Universal Robots PolyScope program: RC_E8_PLACE_831.urp

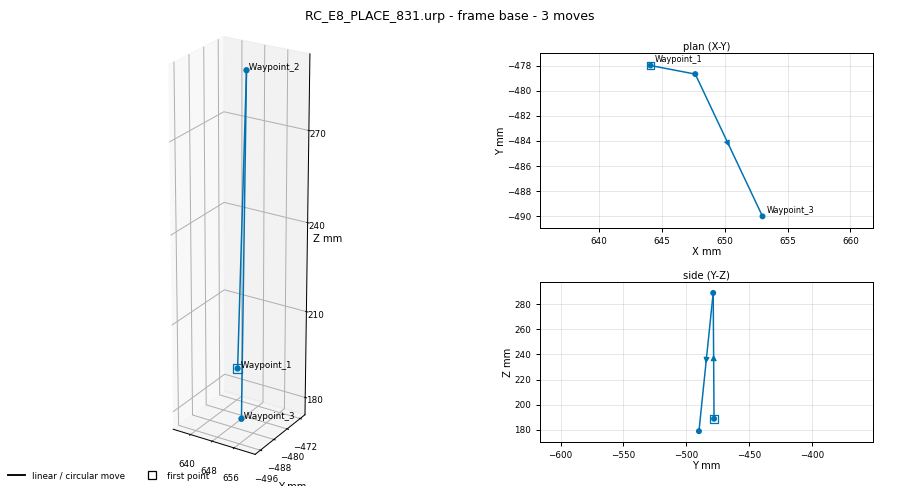
[picture p0: tool path of RC_E8_PLACE_831.urp in frame base, 3 of 3 moves have a stored position in this frame; points joined in program order, loops and branches not executed]
Program RC_E8_PLACE_831 (createdIn=3.0.0 lastSavedIn=3.0.0 directory=/programs installation=default)
Robot Program (runOnlyOnce=true motionType=MoveJ speed=1.047198 acceleration=1.396263 useActiveTCP=false)
  'Program generated by RoboDK v4.1.0 for UR3e_HORNO on 06/09/2022 17:07:52'
  'Using nominal kinematics.'
  'Using Ref. Frame Traslado C: p[0.369000, -0.220000, 0.032000, 0.000000, 0.000000, 0.000000]'
  'Using TCP 0208-0001-0001-307-000-3 Horno: p[0.000000, 0.000000, 0.164750, 0.000000, 0.000000, 0.000000]'
  Script: set_tcp(p[0.000000, 0.000000, 0.164750, 0.000000, 0.000000, 0.000000])
  Script: movej([-0.418006, -2.151118, -0.151320, -2.416408, 1.600991, 4.345870],0.60000,0.12500,0,0.0000)
  MoveL speed 100 mm/s, acceleration 120 mm/s^2 (useActiveTCP=true)
    Waypoint Waypoint_1: TCP in base x=644.083 y=-478 z=188.872 mm, rx=3.1385 ry=-0.0805 rz=-0.0117 rad; joints [-22.639, -103.728, -69.335, -97.291, 89.736, 250.301] deg; flange x=645.315 y=-477.69 z=353.617 mm, rx=3.1385 ry=-0.0805 rz=-0.0117 rad
  'Detach from 0208-0001-0001-307-000-3 Horno'
  MoveL speed 500 mm/s, acceleration 900 mm/s^2 (useActiveTCP=true)
    Waypoint Waypoint_2: TCP in base x=647.647 y=-478.682 z=288.936 mm, rx=-3.1102 ry=0.0802 rz=-0.0087 rad; joints [-23.95, -123.25, -8.67, -138.45, 91.73, 249] deg; flange x=646.6 y=-483.659 z=453.608 mm, rx=-3.1102 ry=0.0802 rz=-0.0087 rad
  Script: movej([-0.418006, -2.151118, -0.151320, -2.416408, 1.600991, 4.345870],0.90000,0.50000,0,0.0000)
  Script: movej([0.453224, -1.802935, -0.994995, -3.455038, 0.479382, 3.143909],0.90000,0.50000,0,0.0000)
  Script: movej([0.434695, -1.947045, -1.926629, -2.377999, 0.460862, 3.124551],0.12000,0.10000,0,0.0000)
  'Attach to 0208-0001-0001-307-000-3 Horno'
  Script: movej([0.453224, -1.802935, -0.994995, -3.455038, 0.479382, 3.143909],0.90000,0.50000,0,0.0000)
  Script: movej([0.420275, -1.803623, -0.993965, -3.453134, 0.446281, 0.000000],0.90000,0.50000,0,0.0000)
  MoveL speed 100 mm/s, acceleration 120 mm/s^2 (useActiveTCP=true)
    Waypoint Waypoint_3: TCP in base x=653 y=-490.005 z=179 mm, rx=1.5841 ry=-0.0094 rz=-0.0052 rad; joints [24.566, -112.37, -109.168, -136.655, 25.106, -1.486] deg; flange x=654.521 y=-325.277 z=181.204 mm, rx=1.5841 ry=-0.0094 rz=-0.0052 rad
  'Detach from 0208-0001-0001-307-000-3 Horno'
  Script: movej([0.420275, -1.803623, -0.993965, -3.453134, 0.446281, 0.000000],0.90000,0.50000,0,0.0000)
